FUNCTION_BLOCK FB_HE_SATT
VAR
END_VAR

END_FUNCTION_BLOCK

(* stored: Version 1.1.0.1
   POU FB_HE_SATT: Id {501a80b3-9bce-49ff-9df4-863a57e47659}, SpecialFunc None *)
